FUNCTION instantexpectedcapVOLT_802L : REAL
VAR_INPUT
	timenow : TIME;
	capacitanceF : REAL;
	PSUratedVoltage : DINT;
	targetVoltage : DINT;
END_VAR
VAR_IN_OUT
	previoustime : REAL;
	Voltlast : REAL;
END_VAR
VAR
	timenowsec : REAL;
	Powerpeak802L : REAL := 9000;
	timestepsec : REAL;
	Ipeak : REAL;
	I : REAL;
END_VAR

(* Function specific to TDK 802L. Must be modified for other models. 
Assumed to using the constant charging and constant power scheme. *)

timenowsec := TIME_TO_REAL(timenow)*0.001;	// From ms to sec
IF PSUratedVoltage = 0 THEN
	instantexpectedcapVOLT_802L := 0;
ELSE
	Ipeak := 2.0*Powerpeak802L/DINT_TO_REAL(PSUratedVoltage);
	timestepsec := timenowsec-previoustime;
	// Return last known voltage if timestep is 0
	IF targetVoltage <= 6000 THEN
		I := Ipeak;
	ELSE
		I := Ipeak*(0.5+(DINT_TO_REAL(PSUratedVoltage)-Voltlast)/DINT_TO_REAL(PSUratedVoltage));
	END_IF
	IF timestepsec >= 0 THEN
		previoustime := previoustime+timestepsec;
		Voltlast := timestepsec/capacitanceF*I+Voltlast;
	END_IF
	IF Voltlast >= DINT_TO_REAL(targetVoltage) THEN
		instantexpectedcapVOLT_802L := DINT_TO_REAL(targetVoltage);
	ELSE
		instantexpectedcapVOLT_802L := Voltlast;
	END_IF;
END_IF

END_FUNCTION

(* stored: Version 1.1.0.1, ProductVersion 3.1.4024.9
   POU instantexpectedcapVOLT_802L: Id {3aeacacb-5011-498a-b5d5-f66866ec9b5a}, SpecialFunc None *)
